FUNCTION_BLOCK SFC4_VIEW (* Composite Function Block Type *)
  (* Standard: 61499-2 *)
  (* Version 0.2, 2003-12-05, JHC, Rockwell Automation, Renamed from NEWCOMPFB. *)
  (* Version 0.1, 2002-01-08, JHC, Rockwell Automation, Added DLY FB as example. *)
  (* Version 0.0, 2000-05-27, JHC, Rockwell Automation *)
  (* Compiler header: package fb.rt.pnp;import fb.rt.vhmi.*; *)
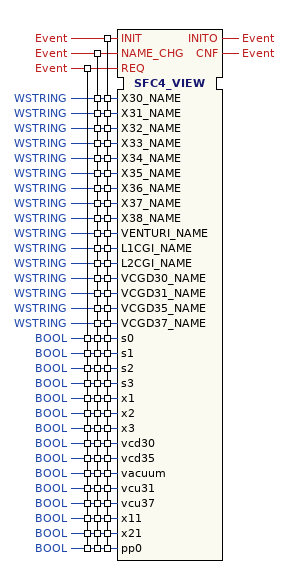
  EVENT_INPUT
    INIT WITH s1, x1, s2, x2, s3, x3, vcd30, vacuum, vcu31, vcu37, x11, x21, s0, pp0, X31_NAME, X32_NAME, X33_NAME, X34_NAME, X35_NAME, X36_NAME, X37_NAME, X38_NAME, VENTURI_NAME, L1CGI_NAME, L2CGI_NAME, X30_NAME, VCGD30_NAME, VCGD31_NAME, VCGD35_NAME, VCGD37_NAME, vcd35; (* Initialization Request *)
    NAME_CHG WITH s1, x1, s2, x2, s3, x3, vcd30, vacuum, vcu31, vcu37, x11, x21, s0, pp0, X31_NAME, X32_NAME, X33_NAME, X34_NAME, X35_NAME, X36_NAME, X37_NAME, X38_NAME, VENTURI_NAME, L1CGI_NAME, L2CGI_NAME, X30_NAME, VCGD30_NAME, VCGD31_NAME, VCGD35_NAME, VCGD37_NAME, vcd35;
    REQ WITH s1, x1, s2, x2, s3, x3, vcd30, vacuum, vcu31, vcu37, x11, x21, s0, pp0, vcd35; (* Normal Execution Request *)
  END_EVENT
  EVENT_OUTPUT
    INITO; (* Initialization Confirm *)
    CNF; (* Execution Confirmation *)
  END_EVENT
  VAR_INPUT
    X30_NAME : WSTRING;
    X31_NAME : WSTRING;
    X32_NAME : WSTRING;
    X33_NAME : WSTRING;
    X34_NAME : WSTRING;
    X35_NAME : WSTRING;
    X36_NAME : WSTRING;
    X37_NAME : WSTRING;
    X38_NAME : WSTRING;
    VENTURI_NAME : WSTRING;
    L1CGI_NAME : WSTRING;
    L2CGI_NAME : WSTRING;
    VCGD30_NAME : WSTRING;
    VCGD31_NAME : WSTRING;
    VCGD35_NAME : WSTRING;
    VCGD37_NAME : WSTRING;
    s0 : BOOL;
    s1 : BOOL;
    s2 : BOOL;
    s3 : BOOL;
    x1 : BOOL;
    x2 : BOOL;
    x3 : BOOL;
    vcd30 : BOOL;
    vcd35 : BOOL;
    vacuum : BOOL;
    vcu31 : BOOL;
    vcu37 : BOOL;
    x11 : BOOL;
    x21 : BOOL;
    pp0 : BOOL;
  END_VAR
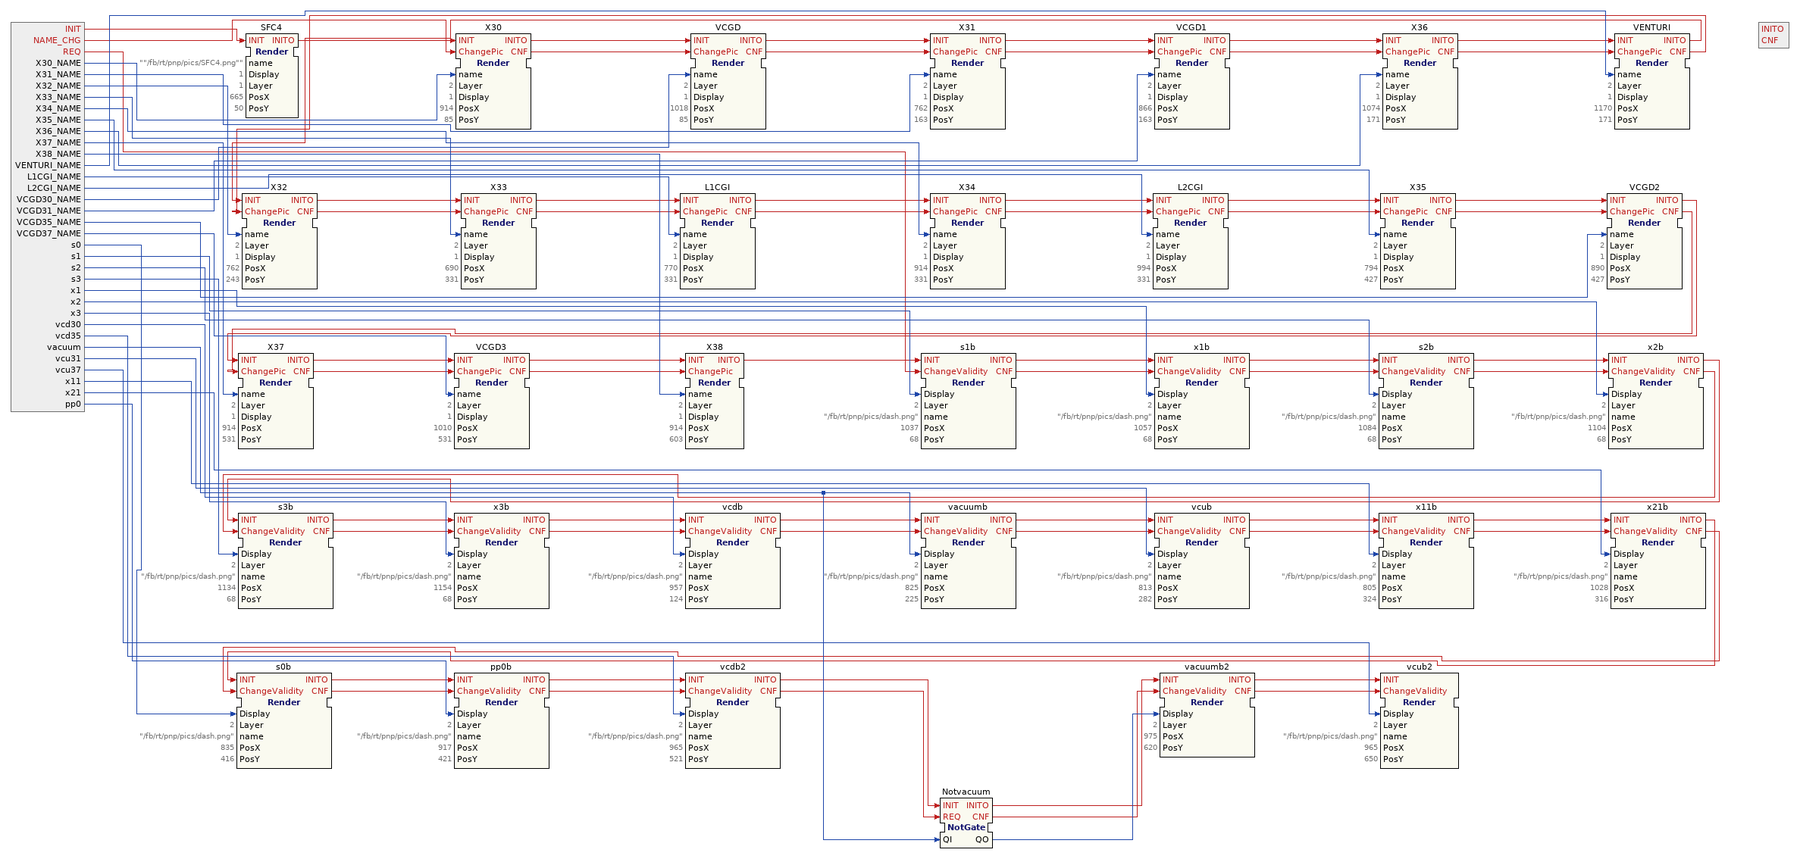
  FBS
    SFC4 : Render(name := ""/fb/rt/pnp/pics/SFC4.png"", Display := 1, Layer := 1, PosX := 665, PosY := 50);
    X30 : Render(Layer := 2, Display := 1, PosX := 914, PosY := 85);
    VCGD : Render(Layer := 2, Display := 1, PosX := 1018, PosY := 85);
    X31 : Render(Layer := 2, Display := 1, PosX := 762, PosY := 163);
    VCGD1 : Render(Layer := 2, Display := 1, PosX := 866, PosY := 163);
    X36 : Render(Layer := 2, Display := 1, PosX := 1074, PosY := 171);
    VENTURI : Render(Layer := 2, Display := 1, PosX := 1170, PosY := 171);
    X32 : Render(Layer := 2, Display := 1, PosX := 762, PosY := 243);
    X33 : Render(Layer := 2, Display := 1, PosX := 690, PosY := 331);
    L1CGI : Render(Layer := 2, Display := 1, PosX := 770, PosY := 331);
    X34 : Render(Layer := 2, Display := 1, PosX := 914, PosY := 331);
    L2CGI : Render(Layer := 2, Display := 1, PosX := 994, PosY := 331);
    X35 : Render(Layer := 2, Display := 1, PosX := 794, PosY := 427);
    VCGD2 : Render(Layer := 2, Display := 1, PosX := 890, PosY := 427);
    X37 : Render(Layer := 2, Display := 1, PosX := 914, PosY := 531);
    VCGD3 : Render(Layer := 2, Display := 1, PosX := 1010, PosY := 531);
    X38 : Render(Layer := 2, Display := 1, PosX := 914, PosY := 603);
    s1b : Render(Layer := 2, name := "/fb/rt/pnp/pics/dash.png", PosX := 1037, PosY := 68);
    x1b : Render(Layer := 2, name := "/fb/rt/pnp/pics/dash.png", PosX := 1057, PosY := 68);
    s2b : Render(Layer := 2, name := "/fb/rt/pnp/pics/dash.png", PosX := 1084, PosY := 68);
    x2b : Render(Layer := 2, name := "/fb/rt/pnp/pics/dash.png", PosX := 1104, PosY := 68);
    s3b : Render(Layer := 2, name := "/fb/rt/pnp/pics/dash.png", PosX := 1134, PosY := 68);
    x3b : Render(Layer := 2, name := "/fb/rt/pnp/pics/dash.png", PosX := 1154, PosY := 68);
    vcdb : Render(Layer := 2, name := "/fb/rt/pnp/pics/dash.png", PosX := 957, PosY := 124);
    vacuumb : Render(Layer := 2, name := "/fb/rt/pnp/pics/dash.png", PosX := 825, PosY := 225);
    vcub : Render(Layer := 2, name := "/fb/rt/pnp/pics/dash.png", PosX := 813, PosY := 282);
    x11b : Render(Layer := 2, name := "/fb/rt/pnp/pics/dash.png", PosX := 805, PosY := 324);
    x21b : Render(Layer := 2, name := "/fb/rt/pnp/pics/dash.png", PosX := 1028, PosY := 316);
    s0b : Render(Layer := 2, name := "/fb/rt/pnp/pics/dash.png", PosX := 835, PosY := 416);
    pp0b : Render(Layer := 2, name := "/fb/rt/pnp/pics/dash.png", PosX := 917, PosY := 421);
    vcdb2 : Render(Layer := 2, name := "/fb/rt/pnp/pics/dash.png", PosX := 965, PosY := 521);
    Notvacuum : NotGate;
    vacuumb2 : Render(Layer := 2, PosX := 975, PosY := 620);
    vcub2 : Render(Layer := 2, name := "/fb/rt/pnp/pics/dash.png", PosX := 965, PosY := 650);
  END_FBS
  EVENT_CONNECTIONS
    SFC4.INITO TO X30.INIT;
    X30.INITO TO VCGD.INIT;
    VCGD.INITO TO X31.INIT;
    X31.INITO TO VCGD1.INIT;
    VCGD1.INITO TO X36.INIT;
    X36.INITO TO VENTURI.INIT;
    VENTURI.INITO TO X32.INIT;
    X32.INITO TO X33.INIT;
    X33.INITO TO L1CGI.INIT;
    L1CGI.INITO TO X34.INIT;
    X34.INITO TO L2CGI.INIT;
    L2CGI.INITO TO X35.INIT;
    X35.INITO TO VCGD2.INIT;
    VCGD2.INITO TO X37.INIT;
    X37.INITO TO VCGD3.INIT;
    VCGD3.INITO TO X38.INIT;
    X38.INITO TO s1b.INIT;
    s1b.INITO TO x1b.INIT;
    x1b.INITO TO s2b.INIT;
    s2b.INITO TO x2b.INIT;
    x2b.INITO TO s3b.INIT;
    s3b.INITO TO x3b.INIT;
    x3b.INITO TO vcdb.INIT;
    vcdb.INITO TO vacuumb.INIT;
    vacuumb.INITO TO vcub.INIT;
    vcub.INITO TO x11b.INIT;
    x11b.INITO TO x21b.INIT;
    x21b.INITO TO s0b.INIT;
    s0b.INITO TO pp0b.INIT;
    pp0b.INITO TO vcdb2.INIT;
    vcdb2.INITO TO Notvacuum.INIT;
    Notvacuum.INITO TO vacuumb2.INIT;
    vacuumb2.INITO TO vcub2.INIT;
    X30.CNF TO VCGD.ChangePic;
    VCGD.CNF TO X31.ChangePic;
    X31.CNF TO VCGD1.ChangePic;
    VCGD1.CNF TO X36.ChangePic;
    X36.CNF TO VENTURI.ChangePic;
    VENTURI.CNF TO X32.ChangePic;
    X32.CNF TO X33.ChangePic;
    X33.CNF TO L1CGI.ChangePic;
    L1CGI.CNF TO X34.ChangePic;
    X34.CNF TO L2CGI.ChangePic;
    L2CGI.CNF TO X35.ChangePic;
    X35.CNF TO VCGD2.ChangePic;
    VCGD2.CNF TO X37.ChangePic;
    X37.CNF TO VCGD3.ChangePic;
    VCGD3.CNF TO X38.ChangePic;
    s1b.CNF TO x1b.ChangeValidity;
    x1b.CNF TO s2b.ChangeValidity;
    s2b.CNF TO x2b.ChangeValidity;
    x2b.CNF TO s3b.ChangeValidity;
    s3b.CNF TO x3b.ChangeValidity;
    x3b.CNF TO vcdb.ChangeValidity;
    vcdb.CNF TO vacuumb.ChangeValidity;
    vacuumb.CNF TO vcub.ChangeValidity;
    vcub.CNF TO x11b.ChangeValidity;
    x11b.CNF TO x21b.ChangeValidity;
    x21b.CNF TO s0b.ChangeValidity;
    s0b.CNF TO pp0b.ChangeValidity;
    pp0b.CNF TO vcdb2.ChangeValidity;
    vcdb2.CNF TO Notvacuum.REQ;
    Notvacuum.CNF TO vacuumb2.ChangeValidity;
    vacuumb2.CNF TO vcub2.ChangeValidity;
    INIT TO SFC4.INIT;
    NAME_CHG TO X30.ChangePic;
    REQ TO s1b.ChangeValidity;
  END_CONNECTIONS
  DATA_CONNECTIONS
    X30_NAME TO X30.name;
    VCGD30_NAME TO VCGD.name;
    X31_NAME TO X31.name;
    VCGD31_NAME TO VCGD1.name;
    X36_NAME TO X36.name;
    VENTURI_NAME TO VENTURI.name;
    X32_NAME TO X32.name;
    L1CGI_NAME TO L1CGI.name;
    X34_NAME TO X34.name;
    L2CGI_NAME TO L2CGI.name;
    X35_NAME TO X35.name;
    VCGD35_NAME TO VCGD2.name;
    X37_NAME TO X37.name;
    VCGD37_NAME TO VCGD3.name;
    X38_NAME TO X38.name;
    s1 TO s1b.Display;
    x1 TO x1b.Display;
    s2 TO s2b.Display;
    x2 TO x2b.Display;
    s3 TO s3b.Display;
    x3 TO x3b.Display;
    vcd30 TO vcdb.Display;
    vacuum TO vacuumb.Display;
    vcu31 TO vcub.Display;
    x11 TO x11b.Display;
    x21 TO x21b.Display;
    s0 TO s0b.Display;
    pp0 TO pp0b.Display;
    vacuum TO Notvacuum.QI;
    X33_NAME TO X33.name;
    Notvacuum.QO TO vacuumb2.Display;
    vcd35 TO vcdb2.Display;
    vcu37 TO vcub2.Display;
  END_CONNECTIONS
END_FUNCTION_BLOCK
